ABB RobotStudio station: CircularPlateWelding_20211129-181223.rsstn

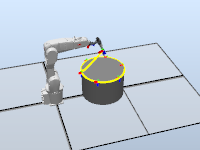
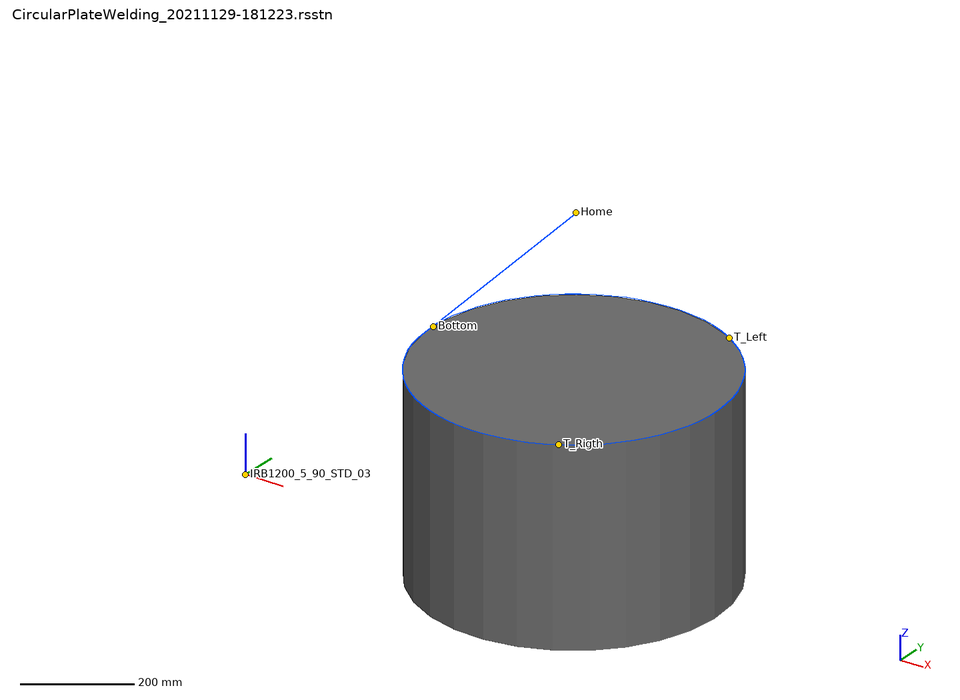
[picture v1: parts stored in the station drawn from their meshes, with robot base, taught points and paths (robot models come from the ABB library and are not in the file)]
Station CircularPlateWelding (saved by RobotStudio 21.3.9648.0)
Controller Controller1
  mechanical unit ROB_1: IRB1200_5_90_STD_03, 6 joints, base frame (0, 0, 0) mm
Layout (positions relative to the parent item):
  - IRB1200_5_90_STD_03 [mechanism, from Robots\IRB1200_5_90_STD_03.rslib] at (0, 0, 0) mm; joint values [0, 0, 0, 0, 0.5236, 0] (rad or m)
  - MyTool [mechanism, from Training Objects\myTool.rslib] at (522.01, 0, 848.1) mm, rotated rx 180 ry 60 rz 180 deg
  - Part_2 [part] at (700, 0, 0) mm, size 600 x 599.1 x 400 mm
Attachment: MyTool is attached to IRB1200_5_90_STD_03 / Link6
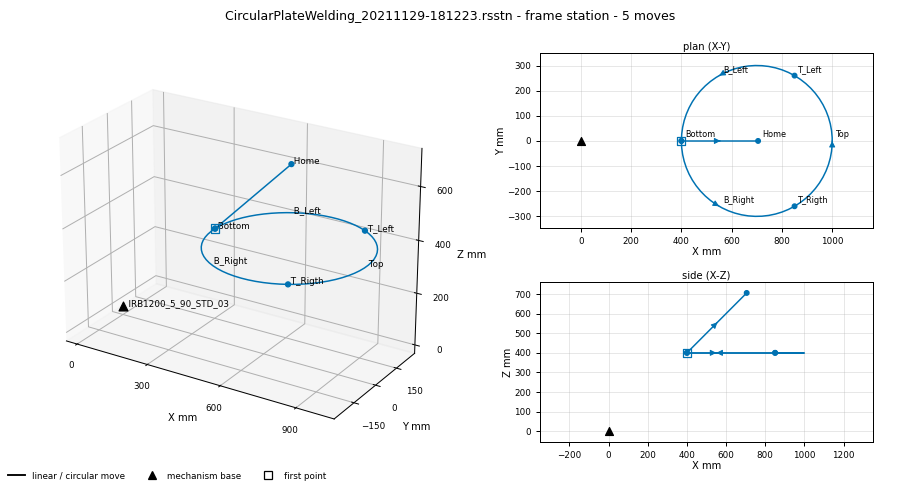
[picture p0: tool path of CircularPlateWelding_20211129-181223.rsstn in frame station, 5 of 5 moves have a stored position in this frame; points joined in program order, loops and branches not executed]
Targets, tools, work objects and paths stored in the station, written as RAPID:
! task T_ROB1
MODULE CalibData
  PERS tooldata MyTool:=[TRUE,[[31.792631019,0,229.638935148],[0.945518576,0,0.325568154,0]],[1,[0,0,1],[1,0,0,0],0,0,0]];
ENDMODULE

! task T_ROB1
MODULE Module1
  CONST robtarget Top:=[[1000,0,400],[0,0,1,0],[-1,0,-1,0],[9E+09,9E+09,9E+09,9E+09,9E+09,9E+09]];
  CONST robtarget T_Left:=[[850,259.807621135,400],[0,0.043619386,0.999048222,0],[0,-1,0,0],[9E+09,9E+09,9E+09,9E+09,9E+09,9E+09]];
  CONST robtarget B_Left:=[[550,259.807621135,400],[0,-0.087155744,0.996194698,0],[0,-1,0,0],[9E+09,9E+09,9E+09,9E+09,9E+09,9E+09]];
  CONST robtarget Bottom:=[[400,0,400],[0,0,1,0],[0,-1,0,0],[9E+09,9E+09,9E+09,9E+09,9E+09,9E+09]];
  CONST robtarget B_Right:=[[550,-259.807621135,400],[0,0.087155743,0.996194698,0],[-1,0,-1,0],[9E+09,9E+09,9E+09,9E+09,9E+09,9E+09]];
  CONST robtarget T_Rigth:=[[850,-259.807621135,400],[0,-0.087155742,0.996194698,0],[-1,0,-1,0],[9E+09,9E+09,9E+09,9E+09,9E+09,9E+09]];
  CONST robtarget Home:=[[704.990919137,0,705.74730631],[0.190808996,0,0.981627183,0],[-1,0,-1,0],[9E+09,9E+09,9E+09,9E+09,9E+09,9E+09]];
  PROC Path_10()
    MoveL Bottom,v1000,z100,MyTool\WObj:=wobj0;
    MoveC B_Right,T_Rigth,v1000,z100,MyTool\WObj:=wobj0;
    MoveC Top,T_Left,v1000,z100,MyTool\WObj:=wobj0;
    MoveC B_Left,Bottom,v1000,z100,MyTool\WObj:=wobj0;
    MoveL Home,v1000,z100,MyTool\WObj:=wobj0;
  ENDPROC
ENDMODULE

